# EPICS substitutions: dpu3/Db/dpu3-v1.substitutions
file "dpu3-det.template" { pattern
{P      DET     ADDR    SCAN    VER}
{$(P)	$(DET1)	0	$(SCAN)	$(PROT_VER)}
{$(P)	$(DET2)	1	$(SCAN)	$(PROT_VER)}
{$(P)	$(DET3)	2	$(SCAN)	$(PROT_VER)}
{$(P)	$(DET4)	3	$(SCAN)	$(PROT_VER)}
}

file "dpu3-gen.template" { pattern
{P      SCAN    VER}
{$(P)	$(SCAN)	$(PROT_VER)}
}
